FUNCTION projArray0 : BOOL
VAR_INPUT
	arr: ARRAY[0..2] OF BOOL;
	idx: DINT;
END_VAR

projArray0 := arr[normProjIdx(idx, 3)];

END_FUNCTION

(* stored: Version 1.1.0.1, ProductVersion 3.1.4022.18
   POU projArray0: Id {b654e354-da2c-4455-9c27-53dde1defc41}, SpecialFunc None *)
